(*
SPDX-FileCopyrightText: © 2026 Oleksandr Tiutyk <trofimich@gmail.com>
SPDX-License-Identifier: MIT
License: https://opensource.org/license/mit
*)

(*!
<summary>Reports a required field or property that the caller considers unspecified.</summary>
<description>
The caller detects the member error; Throw records diagnostics rather than inspecting the object. Dynamic
instances and clones belong to the current task memory manager until cleanup.
</description>
*)
INTERFACE IDataMemberNotSpecifiedException EXTENDS IGeneralException

(*!
<summary>Formats the rejected member and propagates the exception.</summary>
<description>
Call in the owning cyclic task, not during FB_init. Builds a member diagnostic and captures source and
timestamps with zero error code and no inner cause. Input storage is not retained. Allocation failure uses the
shared terminal memory mechanism.
</description>
<param name="dataMemberName">Name of the field or property rejected by the caller.</param>
*)
METHOD Throw
VAR_INPUT
	sourceNamespaceName : STRING;
	sourceClassName : STRING;
	sourcePOUName : STRING;
	sourcePosition : STRING;
	dataMemberName : STRING;
END_VAR
END_METHOD

END_INTERFACE

(* stored: Version 1.1.0.1
   Itf IDataMemberNotSpecifiedException: Id {2350b160-aedd-4da5-961b-4f214e2e1cd3}
   Method Throw: Id {f32c598e-d35c-4a9c-a210-c8741838f001} *)
